PROGRAM pouS6Alarms
VAR
	idbMsgAlarm: FB_CheckMessageBounds;

END_VAR

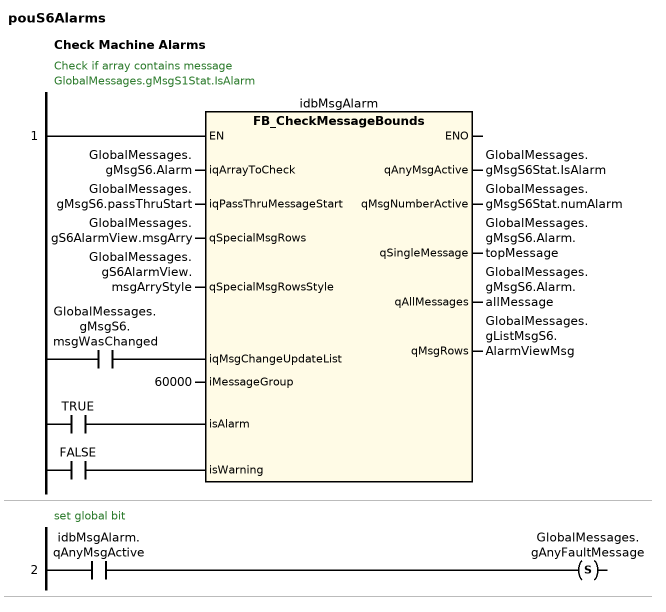
// NETWORK 1: Check Machine Alarms
// Check if array contains message
//
// GlobalMessages.gMsgS1Stat.IsAlarm
idbMsgAlarm(
    iqArrayToCheck := GlobalMessages.gMsgS6.Alarm,
    iqPassThruMessageStart := GlobalMessages.gMsgS6.passThruStart,
    qSpecialMsgRows := GlobalMessages.gS6AlarmView.msgArry,
    qSpecialMsgRowsStyle := GlobalMessages.gS6AlarmView.msgArryStyle,
    iqMsgChangeUpdateList := GlobalMessages.gMsgS6.msgWasChanged,
    iMessageGroup := 60000,
    isAlarm := TRUE,
    isWarning := FALSE,
    qAnyMsgActive => GlobalMessages.gMsgS6Stat.IsAlarm,
    qMsgNumberActive => GlobalMessages.gMsgS6Stat.numAlarm,
    qSingleMessage => GlobalMessages.gMsgS6.Alarm.topMessage,
    qAllMessages => GlobalMessages.gMsgS6.Alarm.allMessage,
    qMsgRows => GlobalMessages.gListMsgS6.AlarmViewMsg); // FB_CheckMessageBounds

// NETWORK 2
// set global bit
GlobalMessages.gAnyFaultMessage S= idbMsgAlarm.qAnyMsgActive;

END_PROGRAM

(* stored: Version 1.1.0.1, ProductVersion 3.1.4024.12
   POU pouS6Alarms: Id {eb79deb6-216d-4dca-ab86-2d4bfd70047a}, SpecialFunc None *)
